TYPE T_CodeBATCH : STRING[10];
END_TYPE

(* stored: Version 1.1.0.1
   DUT T_CodeBATCH: Id {b2264299-582f-4e68-9fb2-da092f7d784c} *)
